{attribute 'qualified_only'}
VAR_GLOBAL
	
automatic : BOOL ;
	CNT_nappilaskuri: INT := 0;
	TEMP_HI_LIMIT: INT := 270;
	TEMP_LO_LIMIT: INT := 242;
	aLampo: ARRAY[1..10] OF INT;
END_VAR

(* stored: Version 1.1.0.1, ProductVersion 3.1.4024.10
   GVL ui: Id {b0f729a2-bd1f-4888-85f4-c0087e171d2a} *)
